PROGRAM MAIN
VAR
END_VAR

Prg_ModbusMasterApplication();

END_PROGRAM

(* stored: Version 1.1.0.1, ProductVersion 3.1.4022.3
   POU MAIN: Id {f34a19a5-5aaa-4615-8f36-da8a3550636a}, SpecialFunc None *)
